{attribute 'qualified_only'}
VAR_GLOBAL
	bDigital_Inputs AT %I* : ARRAY[1..8] OF BOOL;
	bDigital_Outputs AT %Q* : ARRAY[1..8] OF BOOL;
	
	singleAxis : AXIS_REF;
	
	fbSA_Reset				: MC_RESET;
	fbSA_Power				: MC_POWER;
	fbSA_Home				: MC_HOME;
	fbSA_Jog				: MC_JOG;
	
	bSA_ResetExe			: BOOL;
	bSA_PowerEnCmd			: BOOL;
	bSA_PowerEnPositive		: BOOL;
	bSA_PowerEnNegative		: BOOL;
	
	bSA_HomeExe				: BOOL;
	bSA_HomeCamInput		: BOOL;
	
	bSA_JogFwd				: BOOL;
	bSA_JogRev				: BOOL;
	
	lrSA_PowerOverride		: LREAL;
	lrSA_HomePosition		: LREAL;
	lrSA_SetPosition		: LREAL;
	lrSA_JogVelocity		: LREAL;
	
	stSA_Reset				: ST_MC_Status;
	stSA_Power				: ST_MC_Status;
	stSA_Home				: ST_MC_Status;
	stSA_SetPosition		: ST_MC_Status;
	stSA_Jog				: ST_MC_Status;
	
END_VAR

(* stored: Version 1.1.0.1, ProductVersion 3.1.4024.12
   GVL GVL_SA: Id {d5fa82fe-a284-4b51-80a9-8ff9bfa33216} *)
